{attribute addProperty BoxType "EK1100-0000-0018"}
{attribute addProperty Id "Beckhoff_EP8xxxEK1122Beckhoff_EP8xxxEK1122_A0772A641648206"}
{attribute addProperty CRC "584598215"}
{attribute addProperty SizeInBites "1648"}
{attribute addProperty SizeInBytes "206"}
TYPE Beckhoff_EP8xxx_22D842C7 EXTENDS EK1100_179A0949 :
STRUCT
	{attribute addProperty Name "Beckhoff_EP8xxxEK1122"}
	Beckhoff_EP8xxxEK1122 : Beckhoff_EP8xxxEK1122_A0772A64;
END_STRUCT
END_TYPE

(* stored: Version 1.2.0.0, ProductVersion 3.1.4024.9
   DUT Beckhoff_EP8xxx_22D842C7: Id {12da4f07-d464-49e2-9862-f2a4a0c8e9f5} *)
